// TwinCAT 3 PLC project PLC1ADS
// ProgramVersion: 3.1.4026.21
// libraries:
//   Tc2_DataExchange, * (Beckhoff Automation GmbH)
//   Tc2_MC2, * (Beckhoff Automation GmbH)
//   Tc2_Standard, * (Beckhoff Automation GmbH)
//   Tc2_System, * (Beckhoff Automation GmbH)
// project tree:
//   DUTs/ ST_motion.TcDUT
//   / PlcTask.TcTTO
//   POUs/ MAIN.TcPOU
// real-time tasks:
//   TASK PlcTask: cycle T#10ms, priority 20, ADS port 350
// motion (NC):
//   TASK NC-Task 1 SAF: cycle T#10ms, priority 4, ADS port 501
//   TASK NC-Task 1 SVB: cycle T#10ms, priority 8, ADS port 511
//   AXIS Axis 1 (id 1)
//     OtherSettings: AllowMotionCmdToSlave=true
//     encoder EncType=1
//     drive DrvType=5
//       Analog: TorqueSetpointScale=10, ScaleFactorActTorque=0.1
//       TimeComp: TaskDelayCycles=1
//     controller CtrType=1
//       CtrPara: PriorControlFactor=1
//         Observer: BandWidth=20
// variable links:
//   PLC1ADS/PLC1ADS Instance <-> NC-Task 1 SAF/Axes/Axis 1
//     PlcTask Inputs/MAIN.Axisref.NcToPlc <-> Outputs/ToPlc
//     PlcTask Outputs/MAIN.Axisref.PlcToNc <-> Inputs/FromPlc

CONFIGURATION PLC1ADS
    RESOURCE PLC ON TwinCAT3
        TASK PlcTask(INTERVAL := T#10ms, PRIORITY := 20);
        PROGRAM MAIN WITH PlcTask : MAIN;
    END_RESOURCE
END_CONFIGURATION

// ---- DUTs/ST_motion.TcDUT
TYPE ST_motion :
STRUCT
	bEnable   : BOOL;
    bStop     : BOOL;
    bMoveRel  : BOOL;
    rVelocity : REAL;
    rDistance : REAL;
END_STRUCT
END_TYPE

// ---- POUs/MAIN.TcPOU
PROGRAM MAIN
VAR
	Axisref 		:AXIS_REF;
	fbMcPower 		: MC_Power;			// enable and override
	fbMcMoverel		: MC_MoveRelative;  // Relative motion
	fbMcStop		: MC_Stop; 

    //ADS Comms Watchdoog
    fbChkWd      : FB_CheckWatchdog;
	nWatchdogRx  : UDINT;
    bCommFault   : BOOL;
	
	bEnable 	:BOOL; //Enable Controller
	bStop		:BOOL;
	bMoveRel	:BOOL;
	rVelocity	:REAL;
	rDistance	:REAL;
END_VAR

//Watchdog 

fbChkWd(
    bEnable       := TRUE,
    tWatchdogTime := T#5S,
    nCnt          := nWatchdogRx
);

bCommFault := fbChkWd.bWatchdog;

IF NOT bCommFault AND nWatchdogRx <> 0 THEN
fbMcPower(
	Axis:= Axisref, 
	Enable:= bEnable, 
	Enable_Positive:=bEnable , 
	Enable_Negative:=bEnable , 
	Override:= 100 );

	fbMcStop(
	Axis:= Axisref , 
	Execute:= bStop , 
	Deceleration:=  , 
	Jerk:= , 
	Options:= , 
	Done=> , 
	Busy=> , 
	Active=> , 
	CommandAborted=> , 
	Error=> , 
	ErrorID=> );
	
	fbMcMoverel(
	Axis:= Axisref, 
	Execute:= bMoveRel, 
	Distance:= rDistance  , 
	Velocity:= rVelocity, 
	Acceleration:= , 
	Deceleration:= , 
	Jerk:= , 
	BufferMode:= , 
	Options:= , 
	Done=> , 
	Busy=> , 
	Active=> , 
	CommandAborted=> , 
	Error=> , 
	ErrorID=> );
END_IF

END_PROGRAM
